Universal Robots PolyScope program: a_full_bow.urp

Program a_full_bow (installation=string_planes directory=/programs/strings createdIn=5.17.3 lastSavedIn=5.17.3 robotSerialNumber=20245501435)
Calibrated DH parameters: a=[0.000154, -0.137004, -0.385524, -0.00002, 0.000092, 0]; d=[0.162441, 211.794786, -230.585024, 18.923638, 0.099786, 0.09951]; alpha=[1.569493, -0.001902, 0.003874, 1.570111, -1.570167, 0]; deltaTheta=[0, -1.242934, 1.056292, 0.186646, 0.000002, 0.000001]
InitVariablesNode
Robot Program (runOnlyOnce=false)
  SuppressedNode
    MoveL speed 250 mm/s, acceleration 1200 mm/s^2 (useActiveTCP=true) feature=Base
      Waypoint Waypoint_1: TCP in base x=336.638 y=773.336 z=103.937 mm, rx=-1.3698 ry=-2.3362 rz=1.327 rad; joints [-127.102, -6.181, 18.995, -50.118, -88.699, -156.884] deg; TCP offset x=28.21 y=-96.107 z=-99.69 mm, rx=0 ry=0 rz=0 rad
      Waypoint Waypoint_4: TCP in base x=379.853 y=618.981 z=171.588 mm, rx=-1.5056 ry=-2.3348 rz=1.3928 rad; joints [-137.275, -33.165, 63.598, -67.747, -99.589, -156.744] deg
      Waypoint Waypoint_5: TCP in base x=401.443 y=618.981 z=241.831 mm, rx=-1.5056 ry=-2.3348 rz=1.3928 rad; joints [-138.359, -36.11, 58.049, -59.378, -100.467, -157.444] deg
      Waypoint Waypoint_6: TCP in base x=312.76 y=793.568 z=126.299 mm, rx=-1.5435 ry=-2.3549 rz=1.3468 rad; joints [-125.643, -7.751, 17.668, -48.747, -90.653, -148.761] deg
      Waypoint Waypoint_1: TCP in base x=336.638 y=773.336 z=103.937 mm, rx=-1.3698 ry=-2.3362 rz=1.327 rad; joints [-127.102, -6.181, 18.995, -50.118, -88.699, -156.884] deg
  MoveL speed 250 mm/s, acceleration 1200 mm/s^2 (useActiveTCP=true) feature=Base
    Waypoint Waypoint_1: TCP in base x=328.806 y=799.655 z=124.142 mm, rx=-1.4337 ry=-2.1075 rz=1.4431 rad; joints [-125.896, 1.758, -0.737, -31.239, -80.757, -152.721] deg
    Waypoint Waypoint_2: TCP in base x=503.945 y=346.409 z=307.545 mm, rx=-1.4458 ry=-2.2061 rz=1.3509 rad; joints [-161.51, -54.161, 82.326, -66.222, -111.767, -174.226] deg
  MoveL speed 250 mm/s, acceleration 1200 mm/s^2 (useActiveTCP=true) feature=Base
    Waypoint Waypoint_2: TCP in base x=503.945 y=346.409 z=307.545 mm, rx=-1.4458 ry=-2.2061 rz=1.3509 rad; joints [-161.51, -54.161, 82.326, -66.222, -111.767, -174.226] deg
    Waypoint Waypoint_1: TCP in base x=328.806 y=799.655 z=124.142 mm, rx=-1.4337 ry=-2.1075 rz=1.4431 rad; joints [-125.896, 1.758, -0.737, -31.239, -80.757, -152.721] deg
  Wait Sleep waitTime=300
  bow_dir := True
  note_dur := 3
  Timer (action=Start) variable(name=timer_1)
  If bow_dir
    MoveL speed 250 mm/s, acceleration 1200 mm/s^2 (useActiveTCP=true) feature=Base
      Waypoint Waypoint_2: TCP in base x=503.945 y=346.409 z=307.545 mm, rx=-1.4458 ry=-2.2061 rz=1.3509 rad; joints [-161.51, -54.161, 82.326, -66.222, -111.767, -174.226] deg
        Until EXPRESSION (allowActions=false) ExpressionBranch=timer_1≟note_dur
  Else 
    MoveL speed 250 mm/s, acceleration 1200 mm/s^2 (useActiveTCP=true) feature=Base
      Waypoint Waypoint_1: TCP in base x=328.806 y=799.655 z=124.142 mm, rx=-1.4337 ry=-2.1075 rz=1.4431 rad; joints [-125.896, 1.758, -0.737, -31.239, -80.757, -152.721] deg
        Until EXPRESSION (allowActions=false) ExpressionBranch=timer_1≟note_dur
  SuppressedNode
    MoveL speed 250 mm/s, acceleration 1200 mm/s^2 (useActiveTCP=true) feature=Base
      Waypoint Waypoint_1: TCP in base x=277.237 y=734.032 z=156.892 mm, rx=1.7389 ry=2.3104 rz=-1.1078 rad; joints [-126.647, -28.123, 54.729, -74.616, -91.964, -141.812] deg; TCP offset x=28.21 y=-96.107 z=-99.69 mm, rx=0 ry=0 rz=0 rad
      Waypoint Waypoint_3: motionParameters(blendRadius=0.05); TCP in base x=335.809 y=527.638 z=230.762 mm, rx=1.7389 ry=2.3104 rz=-1.1078 rad; joints [-141.244, -51.172, 87.867, -86.053, -101.589, -152.842] deg; TCP offset x=28.21 y=-96.107 z=-99.69 mm, rx=0 ry=0 rz=0 rad
      Waypoint Waypoint_2: TCP in base x=393.128 y=325.659 z=303.053 mm, rx=1.7389 ry=2.3104 rz=-1.1078 rad; joints [-160.523, -67.347, 103.242, -90.17, -113.569, -168.748] deg
  Timer (action=Stop) variable=timer_1
  Timer (action=Reset) variable=timer_1
